# EPICS alarm handler configuration: mps_database/bare/alarms/areas/mpln_bpn21_mp01.alhConfig
GROUP NULL MPLN:BPN21:MP01:1
$ALIAS MPS Link Node 85
$GUIDANCE
LTUH MPS
   Group Name: MPLN:BPN21:MP01:1
   Summary PV:  MPLN:BPN21:MP01:1:STATSUMY
$END
CHANNEL  MPLN:BPN21:MP01:1    MPLN:BPN21:MP01:1:MPS_EN_RBV		-----
CHANNEL  MPLN:BPN21:MP01:1    MPLN:BPN21:MP01:1:LC1_MODE_RBV		-----
